TYPE CM_Valve_PAR :
STRUCT
END_STRUCT
END_TYPE

(* stored: Version 1.1.0.1, ProductVersion 3.1.4024.12
   DUT CM_Valve_PAR: Id {adcf27bd-b8f5-40ee-98b0-646e5f2b443f} *)
